% RSLogix 500 project Calibrar.RSS, saved by version 8.30.00.16 %
PROJECT "UNTITLED"    % processor: Bul.1763 MicroLogix 1100 Series B %

PROGRAM FILES
  LAD 2   12 rungs

DATA FILES
  O0 OUTPUT  4 elements
  I1 INPUT  6 elements
  S2 STATUS  66 elements
  B3 BINARY  1 elements
  T4 TIMER  2 elements
  C5 COUNTER  1 elements
  R6 CONTROL  1 elements
  N7 INTEGER  6 elements
  F8 FLOAT  6 elements

LADDER 2
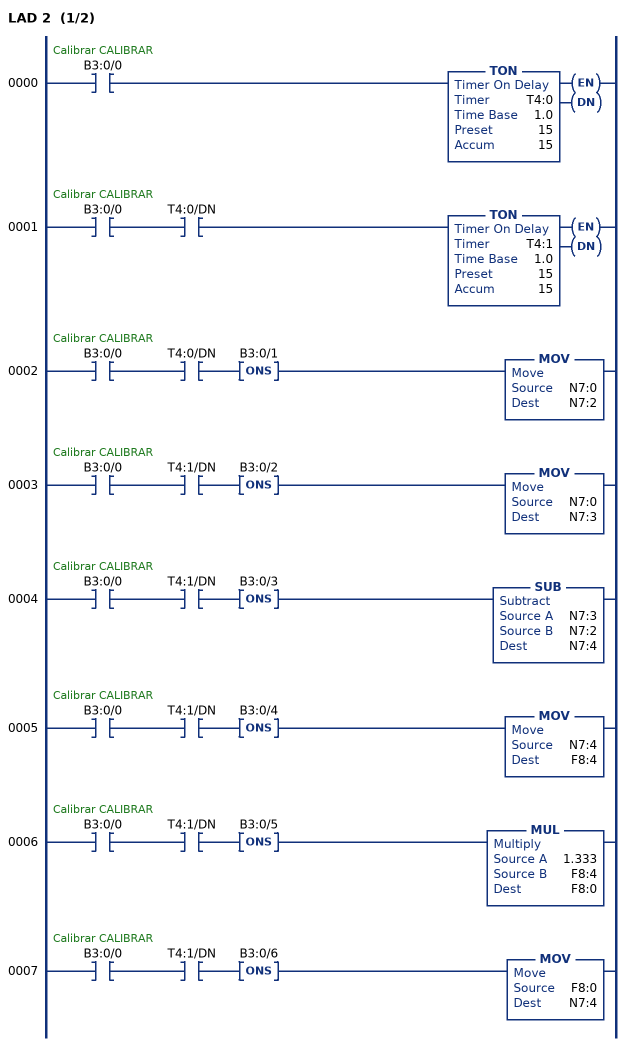
% Rung: 0 %  % edit flag set %
SOR XIC B3:0/0 TON T4:0 1.0 15 15 EOR
%   B3:0/0  CALIBRAR  "Calibrar" %
% Rung: 1 %  % edit flag set %
SOR XIC B3:0/0 XIC T4:0/DN TON T4:1 1.0 15 15 EOR
%   B3:0/0  CALIBRAR  "Calibrar" %
% Rung: 2 %  % edit flag set %
SOR XIC B3:0/0 XIC T4:0/DN ONS B3:0/1 MOV N7:0 N7:2 EOR
%   B3:0/0  CALIBRAR  "Calibrar" %
% Rung: 3 %  % edit flag set %
SOR XIC B3:0/0 XIC T4:1/DN ONS B3:0/2 MOV N7:0 N7:3 EOR
%   B3:0/0  CALIBRAR  "Calibrar" %
% Rung: 4 %  % edit flag set %
SOR XIC B3:0/0 XIC T4:1/DN ONS B3:0/3 SUB N7:3 N7:2 N7:4 EOR
%   B3:0/0  CALIBRAR  "Calibrar" %
% Rung: 5 %  % edit flag set %
SOR XIC B3:0/0 XIC T4:1/DN ONS B3:0/4 MOV N7:4 F8:4 EOR
%   B3:0/0  CALIBRAR  "Calibrar" %
% Rung: 6 %  % edit flag set %
SOR XIC B3:0/0 XIC T4:1/DN ONS B3:0/5 MUL 1.333 F8:4 F8:0 EOR
%   B3:0/0  CALIBRAR  "Calibrar" %
% Rung: 7 %  % edit flag set %
SOR XIC B3:0/0 XIC T4:1/DN ONS B3:0/6 MOV F8:0 N7:4 EOR
%   B3:0/0  CALIBRAR  "Calibrar" %

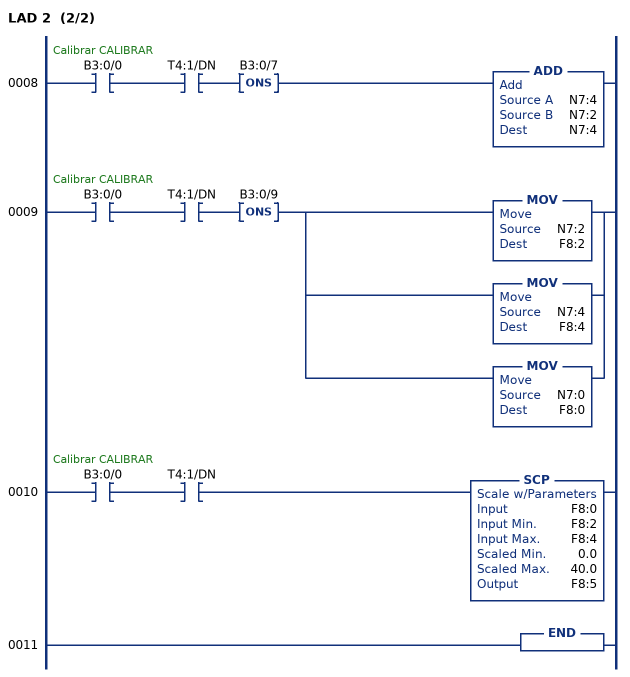
% Rung: 8 %  % edit flag set %
SOR XIC B3:0/0 XIC T4:1/DN ONS B3:0/7 ADD N7:4 N7:2 N7:4 EOR
%   B3:0/0  CALIBRAR  "Calibrar" %
% Rung: 9 %  % edit flag set %
SOR XIC B3:0/0 XIC T4:1/DN ONS B3:0/9 BST MOV N7:2 F8:2 NXB MOV N7:4 F8:4 NXB MOV N7:0 F8:0 BND EOR
%   B3:0/0  CALIBRAR  "Calibrar" %
% Rung: 10 %  % edit flag set %
SOR XIC B3:0/0 XIC T4:1/DN SCP F8:0 F8:2 F8:4 0.0 40.0 F8:5 EOR
%   B3:0/0  CALIBRAR  "Calibrar" %
% Rung: 11 %
SOR END EOR

DATA TABLE (non-zero values as saved)
DATA B3
% B3:0 % 0X02FE
DATA T4
% .PRE .ACC %
% T4:0 % 15 15
% T4:1 % 15 15
DATA N7
% N7:0 % 123 0 30 100 123 33
DATA F8
% F8:0 % 123 nan 30 0 123
% F8:5 % 40
